// TIA Portal V20 export
TYPE "typeSafetyDoorSwitch"
// stored: Access Published, IsFailsafeCompliant true, Namespace Safety
   STRUCT
      SI1_Doorlock : Bool;
      SO1_DoorUnlock : Bool;
      SO2_DoorUnlockReq : Bool;
   END_STRUCT;
END_TYPE
